{attribute 'GeneratedUsingTerminal: EL1502-0000-0001'}
{attribute addProperty BoxType "EL1502-0000-0001"}
{attribute addProperty Id "CNT_InputsAT %I*CNT_Inputs_147BF88E12CNT_OutputsAT %Q*CNT_Outputs_EB14A6758WcStateAT %I*WcState_9091E0EB2InfoDataAT %I*InfoData_32EB74EA10"}
{attribute addProperty CRC "190162306"}
{attribute addProperty Size "32"}
TYPE EL1502_0B55A582 EXTENDS EtcSlaveTerminalBase_947E5A46 :
STRUCT
	{attribute addProperty Name "CNT_Inputs"}
	CNT_Inputs : CNT_Inputs_147BF88E;
	{attribute addProperty Name "CNT_Outputs"}
	CNT_Outputs : CNT_Outputs_EB14A675;
	{attribute addProperty Name "WcState"}
	WcState : WcState_9091E0EB;
	{attribute addProperty Name "InfoData"}
	InfoData : InfoData_32EB74EA;
END_STRUCT
END_TYPE

(* stored: Version 1.2.0.0, ProductVersion 3.1.4024.9
   DUT EL1502_0B55A582: Id {95ff2964-b95a-49fb-9ca8-722b669ac01a} *)
